PROGRAM TESTS_MAIN
VAR
	startTests : BOOL;
END_VAR


IF startTests THEN
	TcUnit.RUN();
END_IF

END_PROGRAM

(* stored: Version 1.1.0.1, ProductVersion 3.1.4024.9
   POU TESTS_MAIN: Id {37444d31-f80d-4c75-941a-8a7910e91182}, SpecialFunc None *)
